(* CODESYS project Simulation_V4.project

Project tree, tasks and I/O mapping:
  Device : CODESYS Virtual Control for Linux SL, CODESYS, order no. 2302000005, version 4.22.0.0
    application Application
      libraries: Standard, 3.5.22.0 (System); VisuDialogs, * (System); Unit Conversion Interfaces, * (Intern); CAA Mathematics, * (CAA Technical Workgroup); SM3_Math, * (CODESYS)
      task MainTask (cyclic, interval t#20ms, priority 1) calls MAIN_PRG, Ablaufkette
      task SoftMotion_PlanningTask (cyclic, interval t#2ms, priority 15) calls nothing
      Kommunikationsverwalter
        OPC UA Server
          Symbolgruppe
      global variables GVL_OPCUA
      visualisation Topics_Vis
      Structs/
        ST_RobotStatus/
          data type ST_RobotStatus
          data type ST_Pose_Axis
          data type ST_Pose_TCP
        ST_RobotAction/
          data type ST_RobotAction
          data type Error_Codes_RobotAction
        ST_RobotCommand/
          data type ST_RobotCommand
          data type ST_Servo_Axis
          data type ST_Servo_TCP
        ST_Orientierung/
          data type ST_euler
          data type ST_quaternions
      old_code/
        data type Manuell_Achse
        data type TCP_Pose
        program PRG_VISU [ST]
        data type JointState
        FB_Robot/
          function block FB_Robot [FBD]
          function block FB_Watchdog [ST]
          function block FB_RobotCommander [ST]
        Interfaces/
          interface IF_RobotStatus: Ist_Pose_Axis, Ist_Pose_TCP, Ist_Mode, Client_Connection_Status, Update_Watchdog
          interface IF_RobotCommand: Soll_Pose_Axis, Soll_Pose_TCP
        function block FB_Roboter [FBD]: Update_Watchdog, Soll_Pose_Axis, Soll_Pose_TCP, Client_Connection_Status, Ist_Mode, Ist_Pose_Axis, Ist_Pose_TCP
        function block Status_POU [ST]
      program MAIN_PRG [FBD]
      FB_Generell/
        function block FB_MoveAction [ST]
        function block FB_Modes [FBD]
        function block FB_RobotStatus [ST]
        function block FB_RobotCommand [ST]
      program Ablaufkette [SFC]
      Funktionen/
        function FUNC_quat_to_euler [ST]
        function block FB_Quat_to_ZYZ [FBD]
        function block FB_ZYZ_to_Quat [FBD]
  libraries: SM3_Robotics, * (CODESYS); VisuSymbols, 4.5.0.0 (System)
  text list GlobalTextList
*)

// Device/Application/old_code/Manuell_Achse
TYPE Manuell_Achse :
STRUCT
	axis_0_plus : BOOL;
	axis_0_minus : BOOL;
	axis_1_plus : BOOL;
	axis_1_minus : BOOL;
	axis_2_plus : BOOL;
	axis_2_minus : BOOL;
	axis_3_plus : BOOL;
	axis_3_minus : BOOL;
	axis_4_plus : BOOL;
	axis_4_minus : BOOL;
	axis_5_plus : BOOL;
	axis_5_minus : BOOL;
	//velocity_spee  einstellen
	//start manuell
END_STRUCT
END_TYPE

// Device/Application/old_code/TCP_Pose
TYPE TCP_Pose :
STRUCT
	trans_x : LREAL;
	trans_y : LREAL;
	trans_z : LREAL;
	rot_x : LREAL;
	rot_y : LREAL;
	rot_z : LREAL;
	rot_w : LREAL;
END_STRUCT
END_TYPE

//TCP Pose in kartesischen Koordinaten
//Rotation wird in quaternions uebermittelt, muss noch umgerechnet werden

// Device/Application/old_code/JointState
TYPE JointState :
STRUCT
	name :ARRAY[0..5] OF STRING;
	position :ARRAY[0..5] OF LREAL; 
	effort :ARRAY[0..5] OF LREAL;
	velocity :ARRAY[0..5] OF LREAL;
END_STRUCT
END_TYPE

// Device/Application/Structs/ST_RobotStatus/ST_RobotStatus
// Gibt den aktuellen Status des Roboters an
TYPE ST_RobotStatus :
STRUCT
	//Joints
	Pos_Axis : ST_Pose_Axis; 	
	
	// TCP mit Orientierung in Quaternions
	Pos_TCP : ST_Pose_TCP;	
	
	//Watchdog
	client_connected : BOOL;
	watchdog_counter : INT;		// Überprüft serverseitige client verbindung
END_STRUCT
END_TYPE

// Device/Application/Structs/ST_RobotCommand/ST_RobotCommand
TYPE ST_RobotCommand :
STRUCT
	// axis manuell
	axis_servo : ST_Servo_Axis;
	
	//tcp manuell
	tcp_servo : ST_Servo_TCP;
	
	//enable: zum starten und stopen der servo_node
	enable : BOOL;
	
	//Watchdog
	client_connected: BOOL;
	watchdog_counter: INT;
END_STRUCT
END_TYPE

// Device/Application/Structs/ST_RobotAction/ST_RobotAction
TYPE ST_RobotAction :
STRUCT
	//Allgemein
	Execute : BOOL;					//Starten der Ausführung (Senden des Goals)
	Error_Code: DINT;				//Feedback ob Ausführung erfolgreich? (Error_code=1)

	//Planer Einstellen
	Motion_Type: STRING;			//string pipeline_id: ompl, pilz_ptp, pilz_lin, pilt_crc
	Planner_ID:STRING;				//string planner_id
	Joint_Goal: BOOL;			
	TCP_GOAL: BOOL;
	num_planning_attempts : DINT;	//int32 num_planning_attempts
	allowed_planning_time: LREAL;	//float64 allowed_planning_time
	max_velocity_scaling: LREAL;		//float64 max_velocity_scaling_factor
	max_acceleration_scaling: LREAL;	//float64 max_acceleration_scaling_factor
	position_tolerance: LREAL;		//float 64 absolute_x_axis_tolerance ->für alle achsen die gleiche toleranz
	orientation_tolerance: LREAL;	//float64
	
	//Joints
	axis_0 : LREAL;		
	axis_1 : LREAL;
	axis_2 : LREAL;
	axis_3 : LREAL;
	axis_4 : LREAL;
	axis_5 : LREAL;
	
	// TCP
	trans_x : LREAL;
	trans_y : LREAL;
	trans_z : LREAL;
	rot_x :  LREAL;
	rot_y : LREAL;
	rot_z : LREAL;
	rot_w : LREAL;
	
	//Watchdog
	client_connected : BOOL;
	watchdog_counter : INT;
END_STRUCT
END_TYPE

// Device/Application/Structs/ST_RobotStatus/ST_Pose_Axis
TYPE ST_Pose_Axis :
STRUCT
	axis_0 : LREAL;
	axis_1 : LREAL;
	axis_2 : LREAL;
	axis_3 : LREAL;
	axis_4 : LREAL;
	axis_5 : LREAL;
END_STRUCT
END_TYPE

// Device/Application/Structs/ST_RobotStatus/ST_Pose_TCP
TYPE ST_Pose_TCP :
STRUCT
	trans_x : LREAL;
	trans_y :  LREAL;
	trans_z : LREAL;
	rot_x : LREAL;
	rot_y : LREAL;
	rot_z : LREAL;
	rot_w : LREAL;
END_STRUCT
END_TYPE

// Device/Application/Structs/ST_RobotCommand/ST_Servo_Axis
TYPE ST_Servo_Axis :
STRUCT
	velocity : LREAL;	
	axis_0 : LREAL;
	axis_1 : LREAL;
	axis_2 : LREAL;
	axis_3 : LREAL;
	axis_4 : LREAL;
	axis_5 : LREAL;
END_STRUCT
END_TYPE

// Device/Application/Structs/ST_RobotCommand/ST_Servo_TCP
TYPE ST_Servo_TCP :
STRUCT
	velocity : LREAL;
	trans_x : LREAL;
	trans_y : LREAL;
	trans_z : LREAL;
	rot_x : LREAL;
	rot_y : LREAL;
	rot_z : LREAL;
	rot_w : LREAL;
END_STRUCT
END_TYPE

// Device/Application/Structs/ST_RobotAction/Error_Codes_RobotAction
{attribute 'qualified_only'}
//{attribute 'strict'}	//CODESYS erlaubt keine TYP Umwandlungen wenn strict aktiv!
{attribute 'to_string'}

TYPE Error_Codes_RobotAction :
(
	NOT_DEFINED := 0,
    SUCCESS := 1,
    FAILURE := 99999,
    PLANNING_FAILED := -1,
    INVALID_MOTION_PLAN := -2,
    MOTION_PLAN_INVALIDATED_BY_ENVIRONMENT_CHANGE := -3,
    CONTROL_FAILED := -4,
    UNABLE_TO_AQUIRE_SENSOR_DATA := -5,
    TIMED_OUT := -6,
    PREEMPTED := -7,
    START_STATE_IN_COLLISION := -10,
    START_STATE_VIOLATES_PATH_CONSTRAINTS := -11,
    START_STATE_INVALID := -26,
    GOAL_IN_COLLISION := -12,
    GOAL_VIOLATES_PATH_CONSTRAINTS := -13,
    GOAL_CONSTRAINTS_VIOLATED := -14,
    GOAL_STATE_INVALID := -27,
    UNRECOGNIZED_GOAL_TYPE := -28,
    INVALID_GROUP_NAME := -15,
    INVALID_GOAL_CONSTRAINTS := -16,
    INVALID_ROBOT_STATE := -17,
    INVALID_LINK_NAME := -18,
    INVALID_OBJECT_NAME := -19,
    FRAME_TRANSFORM_FAILURE := -21,
    COLLISION_CHECKING_UNAVAILABLE := -22,
    ROBOT_STATE_STALE := -23,
    SENSOR_INFO_STALE := -24,
    COMMUNICATION_FAILURE := -25,
    CRASH := -29,
    ABORT := -30,
    NO_IK_SOLUTION := -31
) DINT := NOT_DEFINED;	//Standardwert
END_TYPE

// Device/Application/Structs/ST_Orientierung/ST_euler
//echte Eulerwinkel intrinsich
//ZYZ intrinsisch: bezug auf mitbewegendes Koordinatensystem
//ZYZ extrinsisch: bezug auf festes Koordinatensystem
TYPE ST_euler :
STRUCT
	A : LREAL;	//Z
	B : LREAL;	//Y
	C : LREAL;	//Z
END_STRUCT
END_TYPE

// Device/Application/Structs/ST_Orientierung/ST_quaternions
TYPE ST_quaternions :
STRUCT
	qx: LREAL;
	qy: LREAL;
	qz: LREAL;
	qw: LREAL;
END_STRUCT
END_TYPE

// Device/Application/GVL_OPCUA
{attribute 'qualified_only'}
VAR_GLOBAL
	//Simulation Arm
	
	//Structs global deklarieren!
	RobotAction: ST_RobotAction;	//OPC UA
	Execute : BOOL := FALSE;
	RobotAction_Visu : ST_RobotAction;
	RobotAction_Schrittkette : ST_RobotAction;
	
	RobotStatus : ST_RobotStatus;	//OPC UA
	
	RobotCommand : ST_RobotCommand;	//OPC UA

	
	// Ablaufkette
	TIPP : BOOL; 				// Zum Weiterschalten
	Start_Ablaufkette: BOOL;	// Startet Ablaufkette
	Reset_Ablaufkette: BOOL;	//setzt Schrittkette zurück
	
	//Moveaction 
	Ablauf_HomePos: BOOL;
	Ablauf_Pos1: BOOL;
	Ablauf_Pos2: BOOL;
	Ablauf_Pos3: BOOL;
	Ablauf_Pos4: BOOL;
END_VAR

VAR_GLOBAL CONSTANT
	PI : REAL := 3.14159;
END_VAR

// Device/Application/MAIN_PRG
PROGRAM MAIN_PRG
VAR
///////////////////////////////////////////////////		
	//Modus:
	trig: R_TRIG;

	//Objekt RobotAction
	RobotAction: FB_MoveAction;
	// Actions "initialisieren"
	xMoveHome : BOOL;
	xEx1_ompl_tcp: BOOL;
	xEx2_ompl_joint: BOOL;
	xEx3_pilz_tcp_ptp: BOOL;
	xEx4_pilz_tcp_lin: BOOL;
	
	// ENUM für Error Codes
	Status_Error_Codes_Action : Error_Codes_RobotAction;
///////////////////////////////////////////////////	
	
	//Modes
	Modes: FB_Modes;
	
///////////////////////////////////////////////////		

	// ObjektRobotStatus
	RobotStatus: FB_RobotStatus;
	
///////////////////////////////////////////////////	

	//ObjektRobotCommand
	RobotCommand: FB_RobotCommand;
	VIS_Command_axis_0 : LREAL;
	VIS_Command_axis_1 : LREAL;
	VIS_Command_axis_2 : LREAL;
	VIS_Command_axis_3 : LREAL;
	VIS_Command_axis_4 : LREAL;
	VIS_Command_axis_5 : LREAL;
	VIS_Command_axis_velocity : LREAL;
	
	euler : ST_Euler;
	Status_Quat_to_ZYZ: FB_Quat_to_ZYZ;
	Status_ZYZ_to_Quat : FB_ZYZ_to_Quat;
	Action_zyz_to_quat: FB_ZYZ_to_Quat;
END_VAR

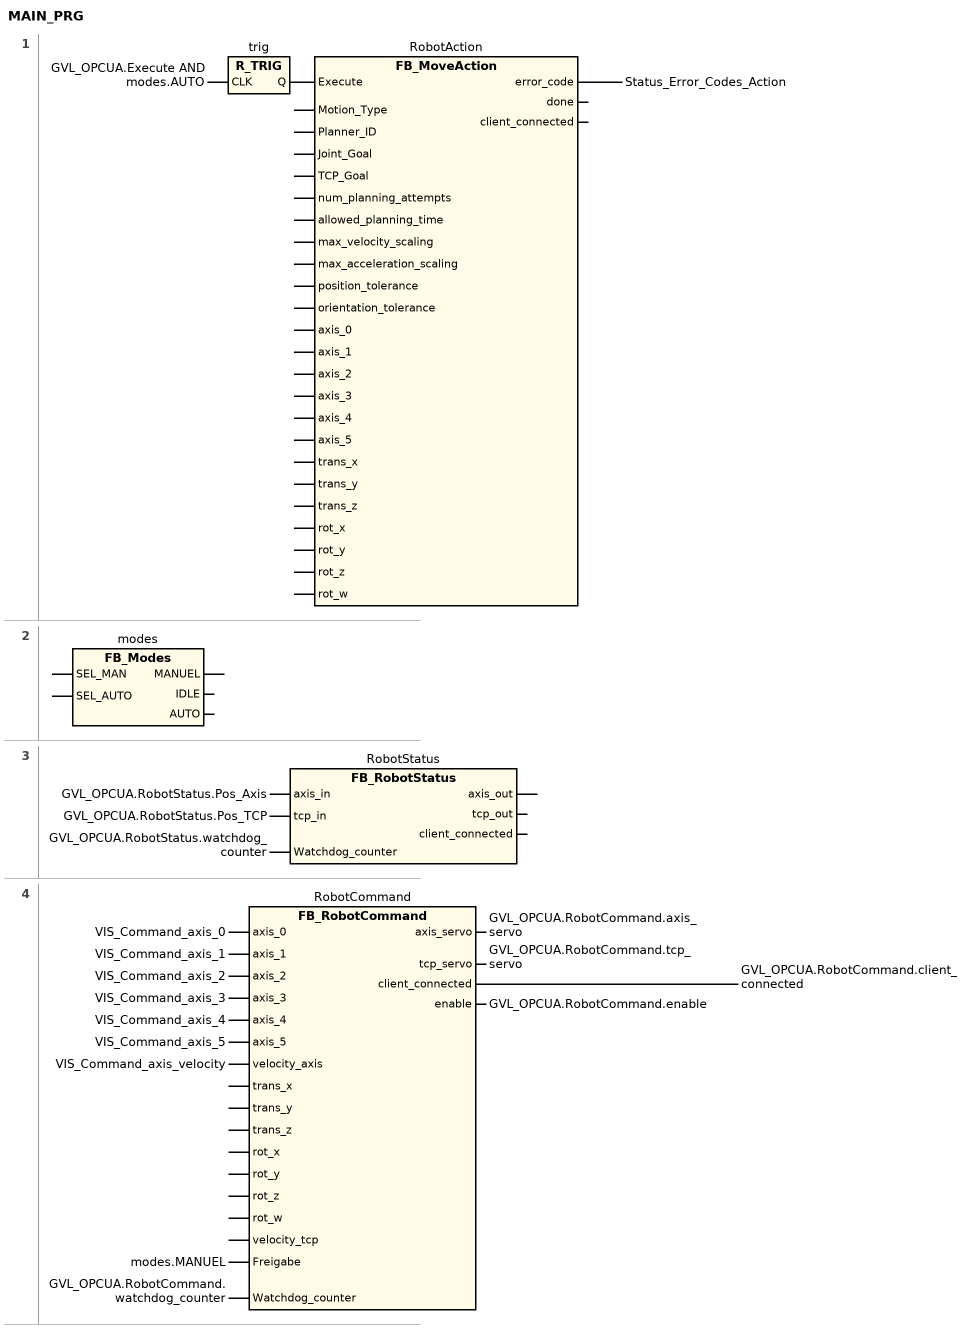
// NETWORK 1
trig(CLK := GVL_OPCUA.Execute AND modes.AUTO); // R_TRIG
RobotAction(Execute := trig.Q); // FB_MoveAction
Status_Error_Codes_Action := RobotAction.error_code;

// NETWORK 2
modes(); // FB_Modes

// NETWORK 3
RobotStatus(
    axis_in := GVL_OPCUA.RobotStatus.Pos_Axis,
    tcp_in := GVL_OPCUA.RobotStatus.Pos_TCP,
    Watchdog_counter := GVL_OPCUA.RobotStatus.watchdog_counter); // FB_RobotStatus

// NETWORK 4
RobotCommand(
    axis_0 := VIS_Command_axis_0,
    axis_1 := VIS_Command_axis_1,
    axis_2 := VIS_Command_axis_2,
    axis_3 := VIS_Command_axis_3,
    axis_4 := VIS_Command_axis_4,
    axis_5 := VIS_Command_axis_5,
    velocity_axis := VIS_Command_axis_velocity,
    Freigabe := modes.MANUEL,
    Watchdog_counter := GVL_OPCUA.RobotCommand.watchdog_counter,
    axis_servo => GVL_OPCUA.RobotCommand.axis_servo,
    tcp_servo => GVL_OPCUA.RobotCommand.tcp_servo,
    enable => GVL_OPCUA.RobotCommand.enable); // FB_RobotCommand
GVL_OPCUA.RobotCommand.client_connected := RobotCommand.client_connected;

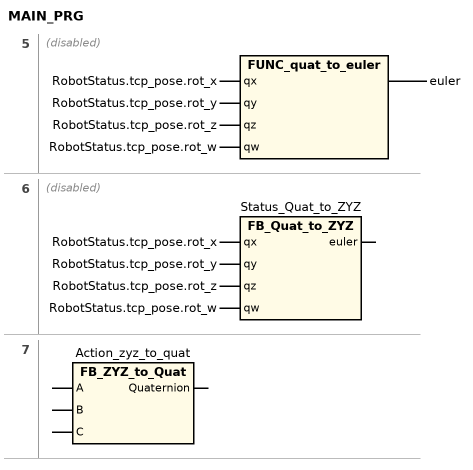
// NETWORK 5 (disabled)
// euler := FUNC_quat_to_euler(qx := RobotStatus.tcp_pose.rot_x, qy := RobotStatus.tcp_pose.rot_y, qz := RobotStatus.tcp_pose.rot_z, qw := RobotStatus.tcp_pose.rot_w);

// NETWORK 6 (disabled)
// Status_Quat_to_ZYZ(
//     qx := RobotStatus.tcp_pose.rot_x,
//     qy := RobotStatus.tcp_pose.rot_y,
//     qz := RobotStatus.tcp_pose.rot_z,
//     qw := RobotStatus.tcp_pose.rot_w); // FB_Quat_to_ZYZ

// NETWORK 7
Action_zyz_to_quat(); // FB_ZYZ_to_Quat

END_PROGRAM

// Device/Application/FB_Generell/FB_MoveAction
FUNCTION_BLOCK FB_MoveAction
VAR_IN_OUT
	RobotAction : ST_RobotAction;
END_VAR
VAR_INPUT
	//wenn modes.auto dann aus VISU schreiben
	//wenn  modes.idle dann aus schrittkette schreiben
	RobotAction_Schrittkette : ST_RobotAction;
	RobotAction_Visu : ST_RobotAction;
	Mode : INT;
	
END_VAR
VAR_OUTPUT

	done : BOOL;
	//Watchdog
	client_connected : BOOL;
END_VAR
VAR
	//Watchdog
	Watchdog_counter : INT;	
	Watchdog_var_old : INT := -1;
	Intervall : TIME :=T#200MS;
	Timer : TON;
	
	//Konvertierung ZYZ->Quat für action
	zyz_to_quat : FB_ZYZ_to_Quat;

END_VAR

// ============================================================
// Auswahl der Quelle
// ============================================================

IF Mode = 0 THEN
    // AUTOMATIK / VISU

    RobotAction.Execute := RobotAction_Visu.Execute;

    RobotAction.Motion_Type := RobotAction_Visu.Motion_Type;
    RobotAction.Planner_ID := RobotAction_Visu.Planner_ID;

    RobotAction.Joint_Goal := RobotAction_Visu.Joint_Goal;
    RobotAction.TCP_GOAL := RobotAction_Visu.TCP_GOAL;

    RobotAction.num_planning_attempts := RobotAction_Visu.num_planning_attempts;
    RobotAction.allowed_planning_time := RobotAction_Visu.allowed_planning_time;
    RobotAction.max_velocity_scaling := RobotAction_Visu.max_velocity_scaling;
    RobotAction.max_acceleration_scaling := RobotAction_Visu.max_acceleration_scaling;
    RobotAction.position_tolerance := RobotAction_Visu.position_tolerance;
    RobotAction.orientation_tolerance := RobotAction_Visu.orientation_tolerance;

    // Joints
    RobotAction.axis_0 := RobotAction_Visu.axis_0;
    RobotAction.axis_1 := RobotAction_Visu.axis_1;
    RobotAction.axis_2 := RobotAction_Visu.axis_2;
    RobotAction.axis_3 := RobotAction_Visu.axis_3;
    RobotAction.axis_4 := RobotAction_Visu.axis_4;
    RobotAction.axis_5 := RobotAction_Visu.axis_5;

    // TCP
    RobotAction.trans_x := RobotAction_Visu.trans_x;
    RobotAction.trans_y := RobotAction_Visu.trans_y;
    RobotAction.trans_z := RobotAction_Visu.trans_z;

    RobotAction.rot_x := RobotAction_Visu.rot_x;
    RobotAction.rot_y := RobotAction_Visu.rot_y;
    RobotAction.rot_z := RobotAction_Visu.rot_z;
    RobotAction.rot_w := RobotAction_Visu.rot_w;


ELSIF Mode = 1 THEN
    // SCHRITTKETTE

    RobotAction.Execute := RobotAction_Schrittkette.Execute;

    RobotAction.Motion_Type := RobotAction_Schrittkette.Motion_Type;
    RobotAction.Planner_ID := RobotAction_Schrittkette.Planner_ID;

    RobotAction.Joint_Goal := RobotAction_Schrittkette.Joint_Goal;
    RobotAction.TCP_GOAL := RobotAction_Schrittkette.TCP_GOAL;

    RobotAction.num_planning_attempts := RobotAction_Schrittkette.num_planning_attempts;
    RobotAction.allowed_planning_time := RobotAction_Schrittkette.allowed_planning_time;
    RobotAction.max_velocity_scaling := RobotAction_Schrittkette.max_velocity_scaling;
    RobotAction.max_acceleration_scaling := RobotAction_Schrittkette.max_acceleration_scaling;
    RobotAction.position_tolerance := RobotAction_Schrittkette.position_tolerance;
    RobotAction.orientation_tolerance := RobotAction_Schrittkette.orientation_tolerance;

    // Joints
    RobotAction.axis_0 := RobotAction_Schrittkette.axis_0;
    RobotAction.axis_1 := RobotAction_Schrittkette.axis_1;
    RobotAction.axis_2 := RobotAction_Schrittkette.axis_2;
    RobotAction.axis_3 := RobotAction_Schrittkette.axis_3;
    RobotAction.axis_4 := RobotAction_Schrittkette.axis_4;
    RobotAction.axis_5 := RobotAction_Schrittkette.axis_5;

    // TCP
    RobotAction.trans_x := RobotAction_Schrittkette.trans_x;
    RobotAction.trans_y := RobotAction_Schrittkette.trans_y;
    RobotAction.trans_z := RobotAction_Schrittkette.trans_z;

    RobotAction.rot_x := RobotAction_Schrittkette.rot_x;
    RobotAction.rot_y := RobotAction_Schrittkette.rot_y;
    RobotAction.rot_z := RobotAction_Schrittkette.rot_z;
    RobotAction.rot_w := RobotAction_Schrittkette.rot_w;

END_IF;


// ============================================================
// OUTPUT
// ============================================================

IF RobotAction.Error_Code = 1 THEN
    done := TRUE;
ELSE
    done := FALSE;
END_IF;



// ============================================================
// Watchdog
// ============================================================

IF RobotAction.watchdog_counter <> Watchdog_var_old THEN
    Watchdog_var_old := RobotAction.watchdog_counter;
    RobotAction.client_connected := TRUE;
    Timer(IN := FALSE);

ELSE
    Timer(
        IN := TRUE,
        PT := Intervall
    );
END_IF;

IF Timer.Q THEN
    RobotAction.client_connected := FALSE;
END_IF;

END_FUNCTION_BLOCK

// Device/Application/Funktionen/FB_ZYZ_to_Quat
FUNCTION_BLOCK FB_ZYZ_to_Quat
VAR_INPUT
	A : LREAL;
	B: LREAL;
	C: LREAL;
END_VAR
VAR_OUTPUT
	Quaternion: SMC_Quat;
END_VAR
VAR
	Rotation_Matrix: SMC_Matrix3;
END_VAR

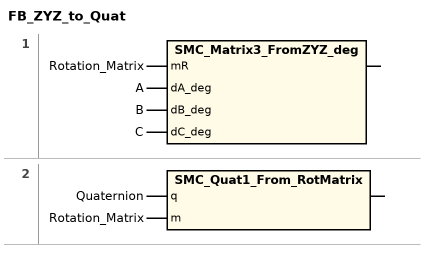
// NETWORK 1
SMC_Matrix3_FromZYZ_deg(mR := Rotation_Matrix, dA_deg := A, dB_deg := B, dC_deg := C);

// NETWORK 2
SMC_Quat1_From_RotMatrix(q := Quaternion, m := Rotation_Matrix);

END_FUNCTION_BLOCK

// Device/Application/FB_Generell/FB_Modes
FUNCTION_BLOCK FB_Modes	//mit Betriebsartenhierachie MAN > AUTO
VAR_INPUT
	SEL_MAN : BOOL;
	SEL_AUTO: BOOL;
END_VAR
VAR_OUTPUT
	MANUEL : BOOL;	//z1
	IDLE: BOOL;		//z0
	AUTO: BOOL;		//z2
END_VAR
VAR
	z0, z1, z2 : BOOL;
	H1, H2: RS;
	z: INT;
END_VAR
VAR // added by the converter: edge detectors and wires of the graphical bodies
    _w1, _w2, _w3 : BOOL;
END_VAR

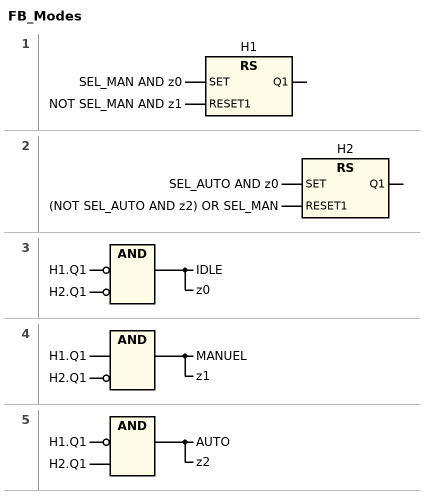
// NETWORK 1
H1(SET := SEL_MAN AND z0, RESET1 := NOT SEL_MAN AND z1); // RS

// NETWORK 2
H2(SET := SEL_AUTO AND z0, RESET1 := (NOT SEL_AUTO AND z2) OR SEL_MAN); // RS

// NETWORK 3
_w1 := NOT H1.Q1 AND NOT H2.Q1;
IDLE := _w1;
z0 := _w1;

// NETWORK 4
_w2 := H1.Q1 AND NOT H2.Q1;
MANUEL := _w2;
z1 := _w2;

// NETWORK 5
_w3 := NOT H1.Q1 AND H2.Q1;
AUTO := _w3;
z2 := _w3;

END_FUNCTION_BLOCK

// Device/Application/FB_Generell/FB_RobotStatus
FUNCTION_BLOCK FB_RobotStatus
VAR_INPUT
	// Axis pose in rad
	axis_in : ST_Pose_Axis;
	
	//TCP Posemit Orientierung in Quaternions
	tcp_in : ST_Pose_TCP;
END_VAR

VAR_IN_OUT
	// Watchdog
	Watchdog_counter : INT;
END_VAR
VAR_OUTPUT
	axis_out : ST_Pose_Axis;
	tcp_out : ST_Pose_TCP;
	client_connected : BOOL;
END_VAR
VAR
	//Watchdog	
	Watchdog_var_old : INT := -1;
	Intervall : TIME :=T#200MS;
	Timer : TON;
END_VAR

//Einbauen ob Ausgabe in RAD ODER GRAD ERFOLGEN SOLL

    axis_out := axis_in;
    tcp_out := tcp_in;

//Watchdog zum Testen ob noch mit StatusClient verbunden!
IF Watchdog_counter <> Watchdog_var_old THEN
	Watchdog_var_old :=  Watchdog_counter;
    client_connected := TRUE;
    Timer(IN := FALSE);

ELSE
    Timer(IN := TRUE,PT := Intervall );
END_IF;

IF Timer.Q THEN
    client_connected := FALSE;
END_IF;

END_FUNCTION_BLOCK

// Device/Application/FB_Generell/FB_RobotCommand
FUNCTION_BLOCK FB_RobotCommand
VAR_INPUT
	axis_0 :LREAL;
	axis_1:LREAL;
	axis_2:LREAL;
	axis_3:LREAL;
	axis_4:LREAL;
	axis_5:LREAL;
	velocity_axis : LREAL;
	
	trans_x:LREAL;
	trans_y:LREAL;
	trans_z:LREAL;
	rot_x:LREAL;
	rot_y:LREAL;
	rot_z:LREAL;
	rot_w:LREAL;
	velocity_tcp: LREAL;
	Freigabe : BOOL;
	enable : BOOL;
END_VAR
VAR_IN_OUT
	Watchdog_counter : INT;	
END_VAR
VAR_OUTPUT
	//globale Variablen damit verknüpfen
	axis_servo : ST_Servo_Axis;
	tcp_servo : ST_Servo_TCP;
	// Watchdog
	client_connected : BOOL;
END_VAR
VAR
	//Watchdog
	Watchdog_var_old : INT := -1;
	Intervall : TIME :=T#200MS;
	Timer : TON;
END_VAR

IF Freigabe THEN

	enable := TRUE;

    axis_servo.axis_0 := axis_0;
    axis_servo.axis_1 := axis_1;
    axis_servo.axis_2 := axis_2;
    axis_servo.axis_3 := axis_3;
    axis_servo.axis_4 := axis_4;
    axis_servo.axis_5 := axis_5;
    axis_servo.velocity := velocity_axis;

    tcp_servo.trans_x := trans_x;
    tcp_servo.trans_y := trans_y;
    tcp_servo.trans_z := trans_z;

    tcp_servo.rot_x := rot_x;
    tcp_servo.rot_y := rot_y;
    tcp_servo.rot_z := rot_z;
    tcp_servo.rot_w := rot_w;

    tcp_servo.velocity := velocity_tcp;

ELSE
	enable := FALSE;

    axis_servo.axis_0 := 0;
    axis_servo.axis_1 := 0;
    axis_servo.axis_2 := 0;
    axis_servo.axis_3 := 0;
    axis_servo.axis_4 := 0;
    axis_servo.axis_5 := 0;
    axis_servo.velocity := 0;

    tcp_servo.trans_x := 0;
    tcp_servo.trans_y := 0;
    tcp_servo.trans_z := 0;

    tcp_servo.rot_x := 0;
    tcp_servo.rot_y := 0;
    tcp_servo.rot_z := 0;
    tcp_servo.rot_w := 0;

    tcp_servo.velocity := 0;

END_IF

//Watchdog zum Testen ob noch mit CommandClient verbunden!
IF Watchdog_counter <> Watchdog_var_old THEN
	Watchdog_var_old :=  Watchdog_counter;
    client_connected := TRUE;
    Timer(IN := FALSE);

ELSE
    Timer(IN := TRUE,PT := Intervall );
END_IF;

IF Timer.Q THEN
    client_connected := FALSE;
END_IF;

END_FUNCTION_BLOCK

// Device/Application/Funktionen/FUNC_quat_to_euler
FUNCTION FUNC_quat_to_euler : ST_euler
VAR_INPUT
	qx : LREAL;
	qy : LREAL;
	qz : LREAL;
	qw : LREAL;
END_VAR
VAR
	r11, r12, r13, r21, r22, r23, r31, r32, r33 : LREAL;
	const_epsilon : LREAL := 1.0E-6; // Toleranz für Gimbal Lock
	result : ST_euler;
	
END_VAR

//Quaternion -> Euler mit ZYZ (intrinsisch) 
//Ausgabe der Euler Winkel in Grad
//Rotationsmatrix Quaternion
r11 := 1.0 - 2.0 * (qy*qy + qz*qz);
r12 := 2.0 * (qx*qy - qz*qw);
r13 := 2.0 * (qx*qz + qy*qw);

r21 := 2.0 * (qx*qy + qz*qw);
r22 := 1.0 - 2.0 * (qx*qx + qz*qz);
r23 := 2.0 * (qy*qz - qx*qw);

r31 := 2.0 * (qx*qz - qy*qw);
r32 := 2.0 * (qy*qz + qx*qw);
r33 := 1.0 - 2.0 * (qx*qx + qy*qy);

result.B := MATH.atan2_func(SQRT(r31*r31+r32*r32),r33);

IF result.B < const_epsilon THEN
	//Gimbal Lock Nordpol
	result.A := 0.0;
	result.C := MATH.atan2_func(r21,r11);
	
ELSIF result.B > (MATH.PI - const_epsilon) THEN
	//Gimbal Lock Südpol
	result.A := 0.0;
	result.C := MATH.atan2_func(-r21,-r11);
ELSE
	//normal
	result.A := MATH.atan2_func(r23,r13);
	result.C := MATH.atan2_func(r32,-r31);
	
END_IF

result.A := result.A * (180.0/MATH.PI);
result.B := result.B * (180.0/MATH.PI);
result.C := result.C * (180.0/MATH.PI);

FUNC_quat_to_euler := result;

END_FUNCTION

// Device/Application/Funktionen/FB_Quat_to_ZYZ
FUNCTION_BLOCK FB_Quat_to_ZYZ
VAR_INPUT
	qx : LREAL;
	qy: LREAL;
	qz:LREAL;
	qw : LREAL;

END_VAR
VAR_OUTPUT
	euler : ST_euler;
END_VAR
VAR
	Quaternion: SMC_Quat;
	Rotation_Matrix: SMC_Matrix3;
END_VAR

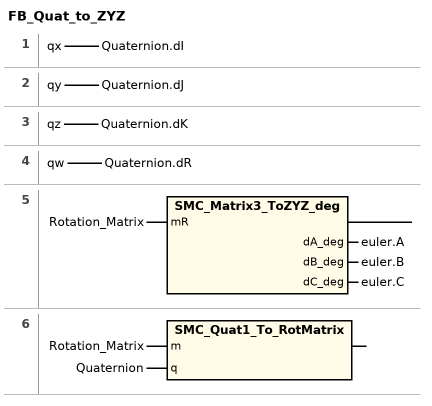
// NETWORK 1
Quaternion.dI := qx;

// NETWORK 2
Quaternion.dJ := qy;

// NETWORK 3
Quaternion.dK := qz;

// NETWORK 4
Quaternion.dR := qw;

// NETWORK 5
SMC_Matrix3_ToZYZ_deg(mR := Rotation_Matrix, dA_deg => euler.A, dB_deg => euler.B, dC_deg => euler.C);

// NETWORK 6
SMC_Quat1_To_RotMatrix(m := Rotation_Matrix, q := Quaternion);

END_FUNCTION_BLOCK

// Device/Application/Ablaufkette
PROGRAM Ablaufkette
VAR
	SFCCurrentStep : STRING;
END_VAR

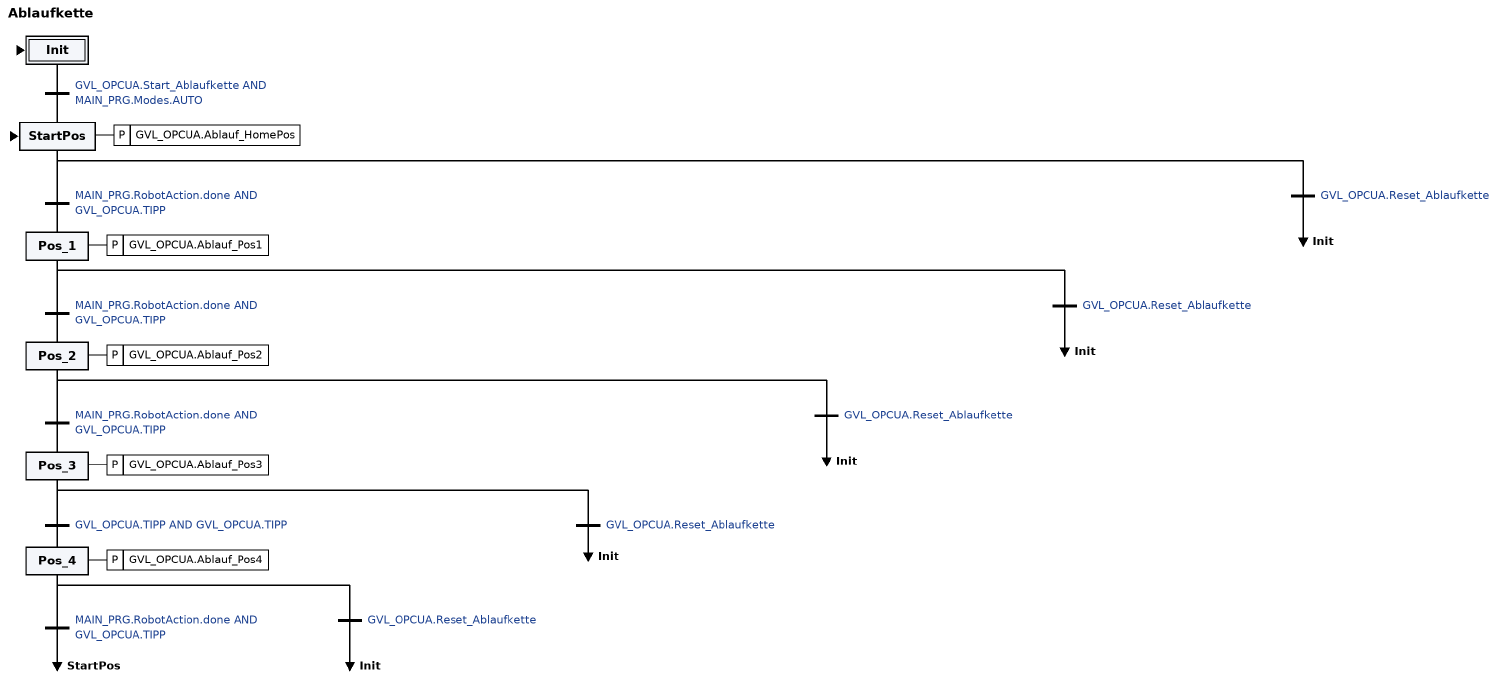
INITIAL_STEP Init:
END_STEP
TRANSITION FROM Init TO StartPos
    := GVL_OPCUA.Start_Ablaufkette AND MAIN_PRG.Modes.AUTO;
END_TRANSITION
STEP StartPos:
    GVL_OPCUA.Ablauf_HomePos(P);
END_STEP
TRANSITION FROM StartPos TO Pos_1
    := MAIN_PRG.RobotAction.done AND GVL_OPCUA.TIPP;
END_TRANSITION
TRANSITION FROM StartPos TO Init
    := GVL_OPCUA.Reset_Ablaufkette;
END_TRANSITION
STEP Pos_1:  // min time t#1s
    GVL_OPCUA.Ablauf_Pos1(P);
END_STEP
TRANSITION FROM Pos_1 TO Pos_2
    := MAIN_PRG.RobotAction.done AND GVL_OPCUA.TIPP;
END_TRANSITION
TRANSITION FROM Pos_1 TO Init
    := GVL_OPCUA.Reset_Ablaufkette;
END_TRANSITION
STEP Pos_2:  // min time t#1s
    GVL_OPCUA.Ablauf_Pos2(P);
END_STEP
TRANSITION FROM Pos_2 TO Pos_3
    := MAIN_PRG.RobotAction.done AND GVL_OPCUA.TIPP;
END_TRANSITION
TRANSITION FROM Pos_2 TO Init
    := GVL_OPCUA.Reset_Ablaufkette;
END_TRANSITION
STEP Pos_3:  // min time t#1s
    GVL_OPCUA.Ablauf_Pos3(P);
END_STEP
TRANSITION FROM Pos_3 TO Pos_4
    := GVL_OPCUA.TIPP AND GVL_OPCUA.TIPP;
END_TRANSITION
TRANSITION FROM Pos_3 TO Init
    := GVL_OPCUA.Reset_Ablaufkette;
END_TRANSITION
STEP Pos_4:  // min time t#1s
    GVL_OPCUA.Ablauf_Pos4(P);
END_STEP
TRANSITION FROM Pos_4 TO StartPos
    := MAIN_PRG.RobotAction.done AND GVL_OPCUA.TIPP;
END_TRANSITION
TRANSITION FROM Pos_4 TO Init
    := GVL_OPCUA.Reset_Ablaufkette;
END_TRANSITION

END_PROGRAM

// Device/Application/old_code/PRG_VISU
PROGRAM PRG_Visu
VAR
    //arrStruct: ARRAY[0..6] OF LREAL;
	Robot : FB_Robot;
	
	//Instanziierung für Roboter
	axis_0_plus :BOOL := FALSE;
	axis_0_minus :BOOL := FALSE;
	axis_1_plus :BOOL := FALSE;
	axis_1_minus :BOOL := FALSE;
	axis_2_plus :BOOL := FALSE;
	axis_2_minus :BOOL := FALSE;
	axis_3_plus :BOOL := FALSE;
	axis_3_minus :BOOL := FALSE;
	axis_4_plus :BOOL := FALSE;
	axis_4_minus :BOOL := FALSE;
	axis_5_plus :BOOL := FALSE;
	axis_5_minus :BOOL := FALSE;
	vis_velocity :LREAL := 0;
END_VAR

Robot();

END_PROGRAM

// Device/Application/old_code/FB_Robot/FB_Robot
FUNCTION_BLOCK FB_Robot
VAR_INPUT
	Command: RobotCommand;
END_VAR
VAR_OUTPUT
	Status: ST_RobotStatus;
END_VAR
VAR
	robotcommand : FB_RobotCommand;
	Watchdog: FB_Watchdog;
END_VAR

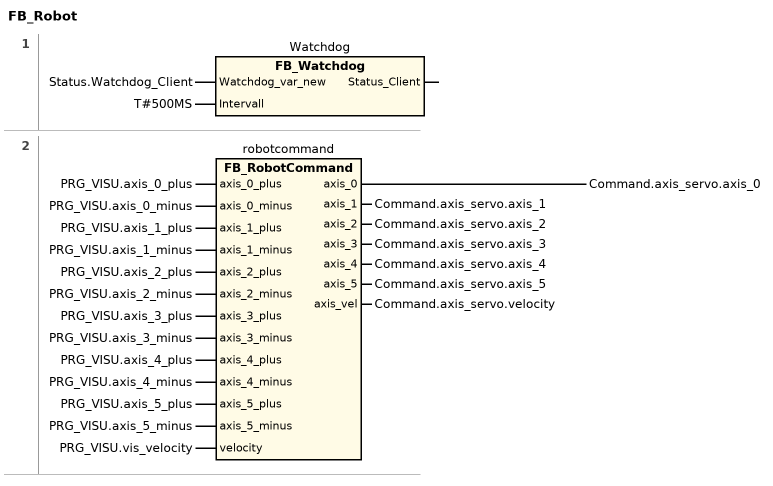
// NETWORK 1
Watchdog(Watchdog_var_new := Status.Watchdog_Client, Intervall := T#500MS); // FB_Watchdog

// NETWORK 2
robotcommand(
    axis_0_plus := PRG_VISU.axis_0_plus,
    axis_0_minus := PRG_VISU.axis_0_minus,
    axis_1_plus := PRG_VISU.axis_1_plus,
    axis_1_minus := PRG_VISU.axis_1_minus,
    axis_2_plus := PRG_VISU.axis_2_plus,
    axis_2_minus := PRG_VISU.axis_2_minus,
    axis_3_plus := PRG_VISU.axis_3_plus,
    axis_3_minus := PRG_VISU.axis_3_minus,
    axis_4_plus := PRG_VISU.axis_4_plus,
    axis_4_minus := PRG_VISU.axis_4_minus,
    axis_5_plus := PRG_VISU.axis_5_plus,
    axis_5_minus := PRG_VISU.axis_5_minus,
    velocity := PRG_VISU.vis_velocity,
    axis_1 => Command.axis_servo.axis_1,
    axis_2 => Command.axis_servo.axis_2,
    axis_3 => Command.axis_servo.axis_3,
    axis_4 => Command.axis_servo.axis_4,
    axis_5 => Command.axis_servo.axis_5,
    axis_vel => Command.axis_servo.velocity); // FB_RobotCommand
Command.axis_servo.axis_0 := robotcommand.axis_0;

END_FUNCTION_BLOCK

// Device/Application/old_code/FB_Robot/FB_Watchdog
FUNCTION_BLOCK FB_Watchdog
VAR_INPUT
	Watchdog_var_new: INT;
	Intervall : TIME;
END_VAR
VAR_OUTPUT
	Status_Client : BOOL;
END_VAR
VAR
	Watchdog_var_old : INT := -1;
	Timer : TON;
END_VAR

IF Watchdog_var_new <> Watchdog_var_old THEN

    Watchdog_var_old := Watchdog_var_new;
    Status_Client := TRUE;
    Timer(IN := FALSE);

ELSE
    Timer(IN := TRUE,PT := Intervall );
END_IF;

IF Timer.Q THEN
    Status_Client := FALSE;
END_IF;

END_FUNCTION_BLOCK

// Device/Application/old_code/FB_Robot/FB_RobotCommander
FUNCTION_BLOCK FB_RobotCommander
VAR_INPUT
	axis_0_plus : BOOL;
	axis_0_minus : BOOL;
	axis_1_plus : BOOL;
	axis_1_minus : BOOL;
	axis_2_plus : BOOL;
	axis_2_minus : BOOL;
	axis_3_plus : BOOL;
	axis_3_minus : BOOL;
	axis_4_plus : BOOL;
	axis_4_minus : BOOL;
	axis_5_plus : BOOL;
	axis_5_minus : BOOL;
	velocity : LREAL;
END_VAR
VAR_OUTPUT
	axis_0 : LREAL;
	axis_1 : LREAL;
	axis_2 : LREAL;
	axis_3 : LREAL;
	axis_4 : LREAL;
	axis_5 : LREAL;
	axis_vel : LREAL;
END_VAR
VAR
END_VAR

// Achse 0
IF axis_0_plus THEN
    axis_0 := 1;
ELSIF axis_0_minus THEN
    axis_0 := -1;
ELSE
    axis_0 := 0;
END_IF;

// Achse 1
IF axis_1_plus THEN
    axis_1 := 1;
ELSIF axis_1_minus THEN
    axis_1 := -1;
ELSE
    axis_1 := 0;
END_IF;

// Achse 2
IF axis_2_plus THEN
    axis_2 := 1;
ELSIF axis_2_minus THEN
    axis_2 := -1;
ELSE
    axis_2 := 0;
END_IF;

// Achse 3
IF axis_3_plus THEN
    axis_3 := 1;
ELSIF axis_3_minus THEN
    axis_3 := -1;
ELSE
    axis_3 := 0;
END_IF;

// Achse 4
IF axis_4_plus THEN
    axis_4 := 1;
ELSIF axis_4_minus THEN
    axis_4 := -1;
ELSE
    axis_4 := 0;
END_IF;

// Achse 5
IF axis_5_plus THEN
    axis_5 := 1;
ELSIF axis_5_minus THEN
    axis_5 := -1;
ELSE
    axis_5 := 0;
END_IF;

// Geschwimdigkeit setzten
axis_vel := velocity;

END_FUNCTION_BLOCK

// Device/Application/old_code/Interfaces/IF_RobotStatus
INTERFACE IF_RobotStatus

PROPERTY Ist_Pose_Axis : ST_Pose_Axis
GET
END_GET
END_PROPERTY

PROPERTY Ist_Pose_TCP : ST_Pose_TCP
GET
END_GET
END_PROPERTY

PROPERTY Ist_Mode : ST_Modes
SET
END_SET
GET
END_GET
END_PROPERTY

PROPERTY Client_Connection_Status : BOOL
SET
END_SET
GET
END_GET
END_PROPERTY

METHOD Update_Watchdog : BOOL
VAR_INPUT
END_VAR
END_METHOD

END_INTERFACE

// Device/Application/old_code/Interfaces/IF_RobotCommand
INTERFACE IF_RobotCommand

PROPERTY Soll_Pose_Axis : ST_Servo_Axis
SET
END_SET
GET
END_GET
END_PROPERTY

PROPERTY Soll_Pose_TCP : ST_Servo_TCP
SET
END_SET
GET
END_GET
END_PROPERTY

END_INTERFACE

// Device/Application/old_code/FB_Roboter
FUNCTION_BLOCK FB_Roboter IMPLEMENTS IF_RobotCommand, IF_RobotStatus
VAR_INPUT
END_VAR
VAR_OUTPUT
END_VAR
VAR
	// --- Command Variablen ---
    _soll_pose_axis : ST_Servo_Axis; // (Passend zu deinem Struct-Namen)
    _soll_pose_tcp  : ST_Servo_TCP;
    
    // --- Status Variablen ---
    _client_connected : BOOL;
    _ist_mode         : ST_Modes;
    _ist_pose_axis    : ST_Pose_Axis;
    _ist_pose_tcp     : ST_Pose_TCP;
END_VAR

// NETWORK 1

{warning 'Methodenimplementierung hinzufügen'}
METHOD Update_Watchdog : BOOL
END_METHOD

{warning 'Eigenschaftenimplementierung hinzufügen'}
PROPERTY Soll_Pose_Axis : ST_Servo_Axis
GET
END_GET
SET
END_SET
END_PROPERTY

{warning 'Eigenschaftenimplementierung hinzufügen'}
PROPERTY Soll_Pose_TCP : ST_Servo_TCP
GET
END_GET
SET
END_SET
END_PROPERTY

{warning 'Eigenschaftenimplementierung hinzufügen'}
PROPERTY Client_Connection_Status : BOOL
GET
END_GET
SET
END_SET
END_PROPERTY

{warning 'Eigenschaftenimplementierung hinzufügen'}
PROPERTY Ist_Mode : ST_Modes
GET
END_GET
SET
END_SET
END_PROPERTY

{warning 'Eigenschaftenimplementierung hinzufügen'}
PROPERTY Ist_Pose_Axis : ST_Pose_Axis
GET
END_GET
SET
END_SET
END_PROPERTY

{warning 'Eigenschaftenimplementierung hinzufügen'}
PROPERTY Ist_Pose_TCP : ST_Pose_TCP
GET
END_GET
SET
END_SET
END_PROPERTY

END_FUNCTION_BLOCK

// Device/Application/old_code/Status_POU
FUNCTION_BLOCK Status_POU
VAR_IN_OUT
END_VAR
VAR_OUTPUT
	Status : ST_RobotStatus;
END_VAR
VAR
END_VAR

END_FUNCTION_BLOCK

// Device/Application/Topics_Vis
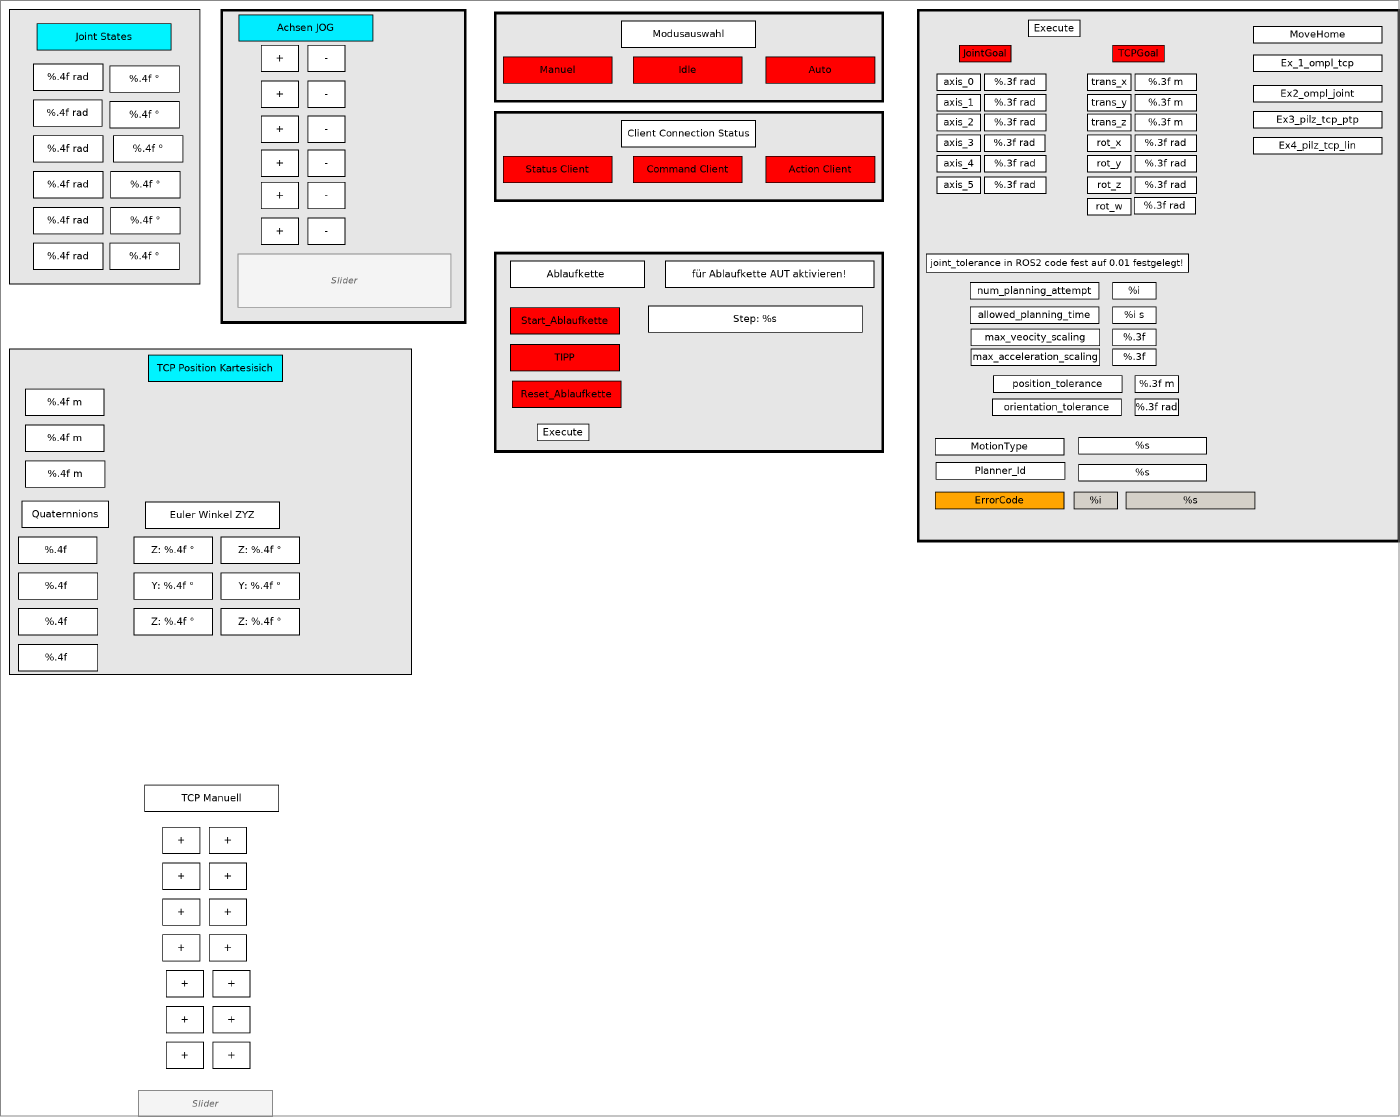
VISUALIZATION Topics_Vis  // 1562x1247
    Rectangle (10,389 449x364)
    Rectangle (246,10 274x351)
    Rectangle (1023,10 539x595)
    Rectangle (551,13 435x101)
    Rectangle (10,10 213x307)
    Rectangle (41,26 150x30), "Joint States"
    Rectangle (165,396 150x30), "TCP Position Kartesisich"
    Rectangle (28,434 88x30), "%.4f m", text variable: MAIN_PRG.RobotStatus.tcp_out.trans_x
    Rectangle (28,474 88x30), "%.4f m", text variable: MAIN_PRG.RobotStatus.tcp_out.trans_y
    Rectangle (28,514 89x30), "%.4f m", text variable: MAIN_PRG.RobotStatus.tcp_out.trans_z
    Rectangle (20,599 88x30), "%.4f", text variable: MAIN_PRG.RobotStatus.tcp_out.rot_x
    Rectangle (20,639 89x30), "%.4f", text variable: MAIN_PRG.RobotStatus.tcp_out.rot_y
    Rectangle (20,679 89x30), "%.4f", text variable: MAIN_PRG.RobotStatus.tcp_out.rot_z
    Rectangle (20,719 89x30), "%.4f", text variable: MAIN_PRG.RobotStatus.tcp_out.rot_w
    Rectangle (291,50 42x30), "+"
        OnMouseDown: execute { MAIN_PRG.VIS_Command_axis_0 := +1; }
        OnMouseUp: execute { MAIN_PRG.VIS_Command_axis_0 := 0; }
    Rectangle (343,50 42x30), "-"
        OnMouseDown: execute { MAIN_PRG.VIS_Command_axis_0 := -1; }
        OnMouseUp: execute { MAIN_PRG.VIS_Command_axis_0 := 0; }
    Rectangle (291,90 42x30), "+"
        OnMouseDown: execute { MAIN_PRG.VIS_Command_axis_1 := +1; }
        OnMouseUp: execute { MAIN_PRG.VIS_Command_axis_1 := 0; }
    Rectangle (343,129 42x30), "-"
        OnMouseDown: execute { MAIN_PRG.VIS_Command_axis_2 := -1; }
        OnMouseUp: execute { MAIN_PRG.VIS_Command_axis_2 := 0; }
    Rectangle (291,129 42x30), "+"
        OnMouseDown: execute { MAIN_PRG.VIS_Command_axis_2 := +1; }
        OnMouseUp: execute { MAIN_PRG.VIS_Command_axis_2 := 0; }
    Rectangle (291,167 42x30), "+"
        OnMouseDown: execute { MAIN_PRG.VIS_Command_axis_3 := +1; }
        OnMouseUp: execute { MAIN_PRG.VIS_Command_axis_3 := 0; }
    Rectangle (343,90 42x30), "-"
        OnMouseDown: execute { MAIN_PRG.VIS_Command_axis_1 := -1; }
        OnMouseUp: execute { MAIN_PRG.VIS_Command_axis_1 := 0; }
    Rectangle (343,167 42x30), "-"
        OnMouseDown: execute { MAIN_PRG.VIS_Command_axis_3 := -1; }
        OnMouseUp: execute { MAIN_PRG.VIS_Command_axis_3 := 0; }
    Rectangle (291,203 42x30), "+"
        OnMouseDown: execute { MAIN_PRG.VIS_Command_axis_4 := +1; }
        OnMouseUp: execute { MAIN_PRG.VIS_Command_axis_4 := 0; }
    Rectangle (343,203 42x30), "-"
        OnMouseDown: execute { MAIN_PRG.VIS_Command_axis_4 := -1; }
        OnMouseUp: execute { MAIN_PRG.VIS_Command_axis_4 := 0; }
    Rectangle (291,243 42x30), "+"
        OnMouseDown: execute { MAIN_PRG.VIS_Command_axis_5 := +1; }
        OnMouseUp: execute { MAIN_PRG.VIS_Command_axis_5 := 0; }
    Rectangle (343,243 42x30), "-"
        OnMouseDown: execute { MAIN_PRG.VIS_Command_axis_5 := -1; }
        OnMouseUp: execute { MAIN_PRG.VIS_Command_axis_5 := 0; }
    Slider (265,283 238x60), variable: MAIN_PRG.VIS_Command_axis_velocity, scale 0..1
    Rectangle (693,23 150x30), "Modusauswahl"
    Rectangle (37,71 78x30), "%.4f rad", text variable: MAIN_PRG.RobotStatus.axis_out.axis_0
    Rectangle (37,111 77x30), "%.4f rad", text variable: MAIN_PRG.RobotStatus.axis_out.axis_1
    Rectangle (37,151 78x30), "%.4f rad", text variable: MAIN_PRG.RobotStatus.axis_out.axis_2
    Rectangle (37,191 78x30), "%.4f rad", text variable: MAIN_PRG.RobotStatus.axis_out.axis_3
    Rectangle (37,231 78x30), "%.4f rad", text variable: MAIN_PRG.RobotStatus.axis_out.axis_4
    Rectangle (37,271 78x30), "%.4f rad", text variable: MAIN_PRG.RobotStatus.axis_out.axis_5
    Rectangle (181,923 42x30), "+"
    Rectangle (181,963 42x30), "+"
    Rectangle (181,1003 42x30), "+"
    Rectangle (181,1043 42x30), "+"
    Rectangle (185,1083 42x30), "+"
    Rectangle (185,1123 42x30), "+"
    Rectangle (185,1163 42x30), "+"
    Rectangle (233,923 42x30), "+"
    Rectangle (233,963 42x30), "+"
    Rectangle (233,1003 42x30), "+"
    Rectangle (233,1043 42x30), "+"
    Rectangle (237,1083 42x30), "+"
    Rectangle (237,1123 42x30), "+"
    Rectangle (237,1163 42x30), "+"
    Slider (154,1217 150x30), scale 0..100
    Rectangle (161,876 150x30), "TCP Manuell"
    Rectangle (266,16 150x30), "Achsen JOG"
    Rectangle (561,63 122x30), "Manuel", colour toggle: MAIN_PRG.Modes.MANUEL
        toggle MAIN_PRG.Modes.SEL_MAN p2164770859=TRUE
    Rectangle (854,63 122x30), "Auto", colour toggle: MAIN_PRG.Modes.AUTO
        toggle MAIN_PRG.Modes.SEL_AUTO p2164770859=TRUE
    Rectangle (706,63 122x30), "Idle", colour toggle: MAIN_PRG.Modes.IDLE
    Rectangle (1045,82 49x19), "axis_0"
    Rectangle (1045,105 49x19), "axis_1"
    Rectangle (1045,127 49x19), "axis_2"
    Rectangle (1045,150 49x19), "axis_3"
    Rectangle (1045,173 49x19), "axis_4"
    Rectangle (1045,197 49x19), "axis_5"
    Rectangle (1098,82 69x19), "%.3f rad", text variable: MAIN_PRG.RobotAction.axis_0
        OnMouseClick: write the text variable via Default
    Rectangle (1098,105 69x19), "%.3f rad", text variable: MAIN_PRG.RobotAction.axis_1
        OnMouseClick: write the text variable via Default
    Rectangle (1098,127 69x19), "%.3f rad", text variable: MAIN_PRG.RobotAction.axis_2
        OnMouseClick: write the text variable via Default
    Rectangle (1098,150 68x19), "%.3f rad", text variable: MAIN_PRG.RobotAction.axis_3
        OnMouseClick: write the text variable via Default
    Rectangle (1098,173 69x19), "%.3f rad", text variable: MAIN_PRG.RobotAction.axis_4
        OnMouseClick: write the text variable via Default
    Rectangle (1098,197 69x19), "%.3f rad", text variable: MAIN_PRG.RobotAction.axis_5
        OnMouseClick: write the text variable via Default
    Rectangle (1213,82 49x19), "trans_x"
    Rectangle (1213,105 49x19), "trans_y"
    Rectangle (1213,127 49x19), "trans_z"
    Rectangle (1213,150 49x19), "rot_x"
    Rectangle (1213,173 49x19), "rot_y"
    Rectangle (1213,197 49x19), "rot_z"
    Rectangle (1266,82 69x19), "%.3f m", text variable: MAIN_PRG.RobotAction.trans_x
        OnMouseClick: write the text variable via Default
    Rectangle (1266,105 69x19), "%.3f m", text variable: MAIN_PRG.RobotAction.trans_y
        OnMouseClick: write the text variable via Default
    Rectangle (1266,127 69x19), "%.3f m", text variable: MAIN_PRG.RobotAction.trans_z
        OnMouseClick: write the text variable via Default
    Rectangle (1266,150 69x19), "%.3f rad", text variable: MAIN_PRG.RobotAction.rot_x
        OnMouseClick: write the text variable via Default
    Rectangle (1266,173 69x19), "%.3f rad", text variable: MAIN_PRG.RobotAction.rot_y
        OnMouseClick: write the text variable via Default
    Rectangle (1266,197 69x19), "%.3f rad", text variable: MAIN_PRG.RobotAction.rot_z
        OnMouseClick: write the text variable via Default
    Rectangle (1213,221 49x19), "rot_w"
    Rectangle (1265,220 69x19), "%.3f rad", text variable: MAIN_PRG.RobotAction.rot_w
        OnMouseClick: write the text variable via Default
    Rectangle (1147,22 58x19), "Execute"
        tap GVL_OPCUA.Execute
    Rectangle (1070,50 58x19), "JointGoal", colour toggle: MAIN_PRG.RobotAction.Joint_Goal
        toggle MAIN_PRG.RobotAction.Joint_Goal
    Rectangle (1241,50 58x19), "TCPGoal", colour toggle: MAIN_PRG.RobotAction.TCP_Goal
        toggle MAIN_PRG.RobotAction.TCP_Goal
    Rectangle (1082,315 144x19), "num_planning_attempt"
    Rectangle (1082,342 144x19), "allowed_planning_time"
    Rectangle (1083,367 144x19), "max_veocity_scaling"
    Rectangle (1083,389 144x19), "max_acceleration_scaling"
    Rectangle (1108,419 144x19), "position_tolerance"
    Rectangle (1107,445 144x19), "orientation_tolerance"
    Rectangle (1241,315 49x19), "%i", text variable: MAIN_PRG.RobotAction.num_planning_attempts
        OnMouseClick: write the text variable via Default
    Rectangle (1241,342 49x19), "%i s", text variable: MAIN_PRG.RobotAction.allowed_planning_time
        OnMouseClick: write the text variable via Default
    Rectangle (1241,367 49x19), "%.3f", text variable: MAIN_PRG.RobotAction.max_velocity_scaling
        OnMouseClick: write the text variable via Default
    Rectangle (1241,389 49x19), "%.3f", text variable: MAIN_PRG.RobotAction.max_acceleration_scaling
        OnMouseClick: write the text variable via Default
    Rectangle (1266,419 49x19), "%.3f m", text variable: MAIN_PRG.RobotAction.position_tolerance
        OnMouseClick: write the text variable via Default
    Rectangle (1266,445 49x19), "%.3f rad", text variable: MAIN_PRG.RobotAction.orientation_tolerance
        OnMouseClick: write the text variable via Default
    Rectangle (1043,489 144x19), "MotionType"
    Rectangle (1044,516 144x19), "Planner_Id"
    Rectangle (1043,549 144x19), "ErrorCode"
    Rectangle (1198,549 49x19), "%i", text variable: MAIN_PRG.RobotAction.error_code
    Rectangle (1203,488 143x19), "%s", text variable: MAIN_PRG.RobotAction.Motion_Type
        OnMouseClick: write the text variable via Default
    Rectangle (1203,518 143x19), "%s", text variable: MAIN_PRG.RobotAction.Planner_ID
        OnMouseClick: write the text variable via Default
    Rectangle (1398,29 144x19), "MoveHome"
        tap MAIN_PRG.xMoveHome
    Rectangle (1256,549 144x19), "%s", text variable: MAIN_PRG.Status_Error_Codes_Action
    Rectangle (551,124 435x101)
    Rectangle (693,134 150x30), "Client Connection Status"
    Rectangle (561,174 122x30), "Status Client", colour toggle: MAIN_PRG.RobotStatus.client_connected
    Rectangle (854,174 122x30), "Action Client", colour toggle: MAIN_PRG.RobotAction.client_connected
    Rectangle (706,174 122x30), "Command Client", colour toggle: MAIN_PRG.RobotCommand.client_connected
    Rectangle (1398,61 144x19), "Ex_1_ompl_tcp"
        tap MAIN_PRG.xEx1_ompl_tcp
    Rectangle (1398,95 144x19), "Ex2_ompl_joint"
        tap MAIN_PRG.xEx2_ompl_joint
    Rectangle (1398,124 144x19), "Ex3_pilz_tcp_ptp"
        tap MAIN_PRG.xEx3_pilz_tcp_ptp
    Rectangle (1398,153 144x19), "Ex4_pilz_tcp_lin"
        tap MAIN_PRG.xEx4_pilz_tcp_lin
    Rectangle (1033,283 293x21), "joint_tolerance in ROS2 code fest auf 0.01 festgelegt!"
    Rectangle (122,73 78x30), "%.4f °", text variable: MAIN_PRG.RobotStatus.axis_out.axis_0 *(180.0/GVL_OPCUA.PI)
    Rectangle (122,113 78x30), "%.4f °", text variable: MAIN_PRG.RobotStatus.axis_out.axis_1 *(180.0/GVL_OPCUA.PI)
    Rectangle (126,151 78x30), "%.4f °", text variable: MAIN_PRG.RobotStatus.axis_out.axis_2 *(180.0/GVL_OPCUA.PI)
    Rectangle (123,191 78x30), "%.4f °", text variable: MAIN_PRG.RobotStatus.axis_out.axis_3 *(180.0/GVL_OPCUA.PI)
    Rectangle (123,231 78x30), "%.4f °", text variable: MAIN_PRG.RobotStatus.axis_out.axis_4 *(180.0/GVL_OPCUA.PI)
    Rectangle (122,271 78x30), "%.4f °", text variable: MAIN_PRG.RobotStatus.axis_out.axis_5 *(180.0/GVL_OPCUA.PI)
    Rectangle (149,599 88x30), "Z: %.4f °", text variable: MAIN_PRG.euler.A
    Rectangle (149,639 88x30), "Y: %.4f °", text variable: MAIN_PRG.euler.B
    Rectangle (149,679 88x30), "Z: %.4f °", text variable: MAIN_PRG.euler.C
    Rectangle (162,560 150x30), "Euler Winkel ZYZ"
    Rectangle (551,281 435x224)
    Rectangle (569,291 150x30), "Ablaufkette"
    Rectangle (569,384 122x30), "TIPP", colour toggle: MAIN_PRG.RobotStatus.client_connected
        tap GVL_OPCUA.TIPP
    Rectangle (569,343 122x30), "Start_Ablaufkette", colour toggle: MAIN_PRG.RobotStatus.client_connected
        tap GVL_OPCUA.Start_Ablaufkette
    Rectangle (723,341 239x30), "Step: %s", text variable: Ablaufkette.SFCCurrentStep
    Rectangle (742,291 233x30), "für Ablaufkette AUT aktivieren!"
    Rectangle (571,425 122x30), "Reset_Ablaufkette", colour toggle: MAIN_PRG.RobotStatus.client_connected
        tap GVL_OPCUA.Reset_Ablaufkette
    Rectangle (599,473 58x19), "Execute"
        tap GVL_OPCUA.Execute
    Rectangle (246,599 88x30), "Z: %.4f °", text variable: MAIN_PRG.Status_Quat_to_ZYZ.euler.A
    Rectangle (246,639 88x30), "Y: %.4f °", text variable: MAIN_PRG.Status_Quat_to_ZYZ.euler.B
    Rectangle (246,679 88x30), "Z: %.4f °", text variable: MAIN_PRG.Status_Quat_to_ZYZ.euler.C
    Rectangle (24,559 97x30), "Quaternnions"
END_VISUALIZATION
